Staubli VAL3: scan_prog.pgx

public program scan_prog(string x_sProg (dimensions=1), string x_sName (dimensions=1))
  local string l_sEmpty
  local num l_nId
begin
  // do the scan and save the file
  // init the sWrite
  call use:stringCopy(l_sEmpty,sWrite)
  // open the file
  nFile=$fileOpen(x_sName+".txt","w")
  // start the scanning
  l_nId=0
  call scanning(x_sProg,0,l_nId,false)
  // save the file
  $fileSet(nFile,sWrite,size(sWrite))
  $fileClose(nFile)
end
